FUNCTION TryConvert_ULINT_TO_UDINT : BOOL
VAR_INPUT
	in : ULINT;
	out : REFERENCE TO UDINT;
END_VAR

IF in > DatatypeLimits.MAX_VALUE_OF_ULINT_WHICH_CAN_BE_HELD_IN_A_UDINT THEN
	RETURN;
END_IF

out := ULINT_TO_UDINT(in);
TryConvert_ULINT_TO_UDINT := TRUE;

END_FUNCTION

(* stored: Version 1.1.0.1, ProductVersion 3.1.4024.12
   POU TryConvert_ULINT_TO_UDINT: Id {171c48d7-2ae7-4be4-a1c0-2bc7415a1511}, SpecialFunc None *)
